TEXTLIST Colors
  1 = '1'
  2 = '2'
  3 = '3'
   = ''
END_TEXTLIST

(* stored: Version 1.1.0.1, ProductVersion 3.1.4018.10
   TextList Colors: Id {893aae36-f63c-430e-ac04-c838b46ccdbf} *)
